(* PLC project Generated.project, CODESYS CODESYS V3.5 SP19 Patch 1 *)
(* stored: creationDateTime 2026-09-01T00:57:57.768470, modificationDateTime 2026-09-01T00:57:57.768470 *)

(* ═══════════════════════════════════════════════════════════════ 🎮 ST_CycleDiveSearchCmd — Sélections IHM cycle plongée (DiveSearch) ═══════════════════════════════════════════════════════════════ *)
TYPE ST_CycleDiveSearchCmd : STRUCT
  TglEnableDiveSearch : BOOL := FALSE;  (* Assistance plongée active *)
  TglBypassDiveSearchSequence : BOOL := FALSE;  (* Bypass séquence DiveSearch *)
  TglBucketAtBottomConfirmed : BOOL := FALSE;  (* Attestation manuelle fond *)
END_STRUCT;
END_TYPE
